FUNCTION Norm_x : REAL
VAR_INPUT
	raw_input : REAL;
	x_max : INT := 32767;
	x_min : INT := 0;
END_VAR
VAR
END_VAR

// 0 - 10V AI INPUT 
Norm_x := (raw_input - x_min) / (x_max - x_min);

END_FUNCTION

(* stored: Version 1.1.0.1, ProductVersion 3.1.4024.11
   POU Norm_x: Id {93db9a71-e368-46de-bb64-aadc328fec0e}, SpecialFunc None *)
